// TIA Portal V19 export
TYPE "lexchangetray_typeroller_signalTM_Cmd_1"
// Type: Bool
// stored: Access Published
   STRUCT
      simActive : Bool;   // Manual mode parameters for axis control interface
   END_STRUCT;
END_TYPE
